// TIA Portal V18 export
DATA_BLOCK "3WayValve_DB"   // DB108
VERSION : 0.1
// stored: AutoNumber true, DBAccessibleFromOPCUA true, DBAccessibleFromWebserver true, InstanceOfName 3WayValve, InstanceOfType FB
"3WayValve"
   // VAR_INPUT
   //    "auto/manual" : Bool;
   //    v1_open_auto : Bool;
   //    v1_open_man : Bool;
   //    v1_fbk_open : Bool;
   //    v1_fbk_close : Bool;
   //    v2_open_auto : Bool;
   //    v2_open_man : Bool;
   //    v2_fbk_open : Bool;
   //    reset : Bool;
   //    intl : Bool;
   //    monito_time : Time;
   //    Mon_En : Bool;
   // END_VAR
   // VAR_OUTPUT
   //    v1_cmd1 : Bool;
   //    v2_cmd2 : Bool;
   //    fault : Bool;
   //    status : Int;
   // END_VAR
   // VAR
   //    open_fault : Bool;
   //    close_fault : Bool;
   //    IEC_Timer_0_Instance : TON_TIME;
   //    IEC_Timer_0_Instance_1 { S7_SetPoint := 'True'} : TON_TIME;
   //    IEC_Timer_0_Instance_2 { S7_SetPoint := 'True'} : TON_TIME;
   //    V1_ON : Bool;
   // END_VAR
BEGIN
END_DATA_BLOCK
